{attribute addProperty BoxType "KL2641"}
{attribute addProperty Id "StateAT %I*BOOL000OutputAT %Q*BOOL000"}
{attribute addProperty CRC "75417483"}
{attribute addProperty SizeInBites "0"}
{attribute addProperty SizeInBytes "0"}
TYPE Channel_047EC78B :
STRUCT
	{attribute addProperty Name "State"}
	State AT %I* : BOOL;
	{attribute addProperty Name "Output"}
	Output AT %Q* : BOOL;
END_STRUCT
END_TYPE

(* stored: Version 1.2.0.0, ProductVersion 3.1.4024.9
   DUT Channel_047EC78B: Id {99a1adcf-decd-4147-bf72-c704260aa882} *)
